(* PLC project mtcs, Institute of Astronomy Onto 0.0.1 *)
(* stored: creationDateTime 2025-03-07T11:57:23.240244, modificationDateTime 2025-03-07T11:57:23.240244 *)

TYPE MTCSParts : STRUCT
  {attribute 'TcHmiSymbol.Show'}
  telemetry : Telemetry;  (* The telemetry *)
  {attribute 'TcHmiSymbol.Show'}
  cover : Cover;  (* The Cover of the telescope *)
  {attribute 'TcHmiSymbol.Show'}
  m1 : M1;  (* The primary mirror of the telescope *)
  {attribute 'TcHmiSymbol.Show'}
  m2 : M2;  (* The secondary mirror of the telescope *)
  {attribute 'TcHmiSymbol.Show'}
  m3 : M3;  (* The tertiary mirror of the telescope *)
  {attribute 'TcHmiSymbol.Show'}
  services : Services;  (* The Services system *)
  {attribute 'TcHmiSymbol.Show'}
  safety : Safety;  (* The safety *)
  {attribute 'TcHmiSymbol.Show'}
  hydraulics : Hydraulics;  (* The hydraulics *)
  {attribute 'TcHmiSymbol.Show'}
  axes : Axes;  (* The axes *)
  {attribute 'TcHmiSymbol.Show'}
  dome : Dome;  (* The dome *)
  {attribute 'TcHmiSymbol.Show'}
  configManager : ConfigManager;  (* The config manager (to load/save/activate configuration data) *)
END_STRUCT;
END_TYPE

TYPE MTCSProcesses : STRUCT
  {attribute 'TcHmiSymbol.Show'}
  initialize : Process;  (* Start initializing the whole MTCS *)
  {attribute 'TcHmiSymbol.Show'}
  lock : Process;  (* Lock the whole MTCS *)
  {attribute 'TcHmiSymbol.Show'}
  unlock : Process;  (* Unlock the whole MTCS *)
  {attribute 'TcHmiSymbol.Show'}
  changeOperator : ChangeOperatorStateProcess;  (* Change the operator (e.g. OBSERVER, TECH, ...) *)
  {attribute 'TcHmiSymbol.Show'}
  verifyPassword : ChangeOperatorStateProcess;  (* Only verify the operator password *)
  {attribute 'TcHmiSymbol.Show'}
  reboot : Process;  (* Reboot the whole MTCS *)
  {attribute 'TcHmiSymbol.Show'}
  shutdown : Process;  (* Shutdown the whole MTCS *)
  {attribute 'TcHmiSymbol.Show'}
  wakeUp : Process;  (* Wake up the whole MTCS *)
  {attribute 'TcHmiSymbol.Show'}
  goToSleep : Process;  (* Let the whole MTCS go to sleep *)
  {attribute 'TcHmiSymbol.Show'}
  stop : Process;  (* Stop the dome and telescope *)
  {attribute 'TcHmiSymbol.Show'}
  endOfNight : Process;  (* End of night *)
  {attribute 'TcHmiSymbol.Show'}
  changeInstrument : MTCSChangeInstrumentProcess;  (* Change the instrument *)
  {attribute 'TcHmiSymbol.Show'}
  point : MTCSPointProcess;  (* Point the telescope and dome to a new target *)
  {attribute 'TcHmiSymbol.Show'}
  emergencyClose : Process;  (* Close the dome and shutter asap *)
  {attribute 'TcHmiSymbol.Show'}
  changeOperatingMode : ChangeOperatingModeStateProcess;  (* Change the operating mode (e.g. LOCAL, REMOTE, ...) *)
  {attribute 'TcHmiSymbol.Show'}
  mocsObservation : MTCSMocsObservationProcess;  (* Notifications about MOCS observation status *)
  {attribute 'TcHmiSymbol.Show'}
  remoteConnectionCheck : Process;  (* Remote connection checking *)
  {attribute 'TcHmiSymbol.Show'}
  remoteConnectionPortCheck : Process;  (* Remote connection port checking *)
  {attribute 'TcHmiSymbol.Show'}
  resetWatchdogTimer : Process;  (* Reset the watchdog timer *)
END_STRUCT;
END_TYPE

TYPE MTCSStatuses : STRUCT
  {attribute 'TcHmiSymbol.Show'}
  initializationStatus : InitializationStatus;
  {attribute 'TcHmiSymbol.Show'}
  healthStatus : HealthStatus;
  {attribute 'TcHmiSymbol.Show'}
  busyStatus : BusyStatus;
  {attribute 'TcHmiSymbol.Show'}
  operatorStatus : OperatorStatus;
  {attribute 'TcHmiSymbol.Show'}
  passwordHealthStatus : HealthStatus;
  {attribute 'TcHmiSymbol.Show'}
  activityStatus : ActivityStatus;
  {attribute 'TcHmiSymbol.Show'}
  operatingModeStatus : OperatingModeStatus;
END_STRUCT;
END_TYPE

TYPE MTCSInstrumentsConfig : STRUCT
  {attribute 'TcHmiSymbol.Show'}
  instrument0 : InstrumentConfig;  (* Instrument 0 *)
  {attribute 'TcHmiSymbol.Show'}
  instrument1 : InstrumentConfig;  (* Instrument 1 *)
  {attribute 'TcHmiSymbol.Show'}
  instrument2 : InstrumentConfig;  (* Instrument 2 *)
  {attribute 'TcHmiSymbol.Show'}
  instrument3 : InstrumentConfig;  (* Instrument 3 *)
  {attribute 'TcHmiSymbol.Show'}
  instrument4 : InstrumentConfig;  (* Instrument 4 *)
  {attribute 'TcHmiSymbol.Show'}
  instrument5 : InstrumentConfig;  (* Instrument 5 *)
  {attribute 'TcHmiSymbol.Show'}
  instrument6 : InstrumentConfig;  (* Instrument 6 *)
  {attribute 'TcHmiSymbol.Show'}
  instrument7 : InstrumentConfig;  (* Instrument 7 *)
  {attribute 'TcHmiSymbol.Show'}
  instrument8 : InstrumentConfig;  (* Instrument 8 *)
  {attribute 'TcHmiSymbol.Show'}
  instrument9 : InstrumentConfig;  (* Instrument 9 *)
END_STRUCT;
END_TYPE

TYPE MTCSEndOfNightStepConfig : STRUCT
  {attribute 'TcHmiSymbol.Show'}
  description : STRING;  (* Description of this step (to show in HMI) *)
  {attribute 'TcHmiSymbol.Show'}
  parkAxes : BOOL;  (* Park the axes *)
  {attribute 'TcHmiSymbol.Show'}
  parkAxesPosition : STRING;  (* Position to park the axes *)
  {attribute 'TcHmiSymbol.Show'}
  parkAxesWait : BOOL;  (* Wait until the axes is parked *)
  {attribute 'TcHmiSymbol.Show'}
  parkM3 : BOOL;  (* Park M3 *)
  {attribute 'TcHmiSymbol.Show'}
  parkM3Position : STRING;  (* Position to park M3 *)
  {attribute 'TcHmiSymbol.Show'}
  parkM3Wait : BOOL;  (* Wait until M3 is parked *)
  {attribute 'TcHmiSymbol.Show'}
  parkDome : BOOL;  (* Park the dome *)
  {attribute 'TcHmiSymbol.Show'}
  parkDomePosition : STRING;  (* Position to park the dome *)
  {attribute 'TcHmiSymbol.Show'}
  parkDomeWait : BOOL;  (* Wait until the dome is parked *)
  {attribute 'TcHmiSymbol.Show'}
  closeCover : BOOL;  (* Close the cover *)
  {attribute 'TcHmiSymbol.Show'}
  closeCoverWait : BOOL;  (* Wait until the cover is closed *)
  {attribute 'TcHmiSymbol.Show'}
  closeDome : BOOL;  (* Close the dome *)
  {attribute 'TcHmiSymbol.Show'}
  closeDomeWait : BOOL;  (* Wait until the dome is closed *)
  {attribute 'TcHmiSymbol.Show'}
  stop : BOOL;  (* Stop the axes and dome *)
  {attribute 'TcHmiSymbol.Show'}
  stopWait : BOOL;  (* Wait until the axes and dome are stopped *)
  {attribute 'TcHmiSymbol.Show'}
  goToSleep : BOOL;  (* Make the telescope go to sleep *)
  {attribute 'TcHmiSymbol.Show'}
  goToSleepWait : BOOL;  (* Wait until the telescope is sleeping *)
END_STRUCT;
END_TYPE

TYPE MTCSEndOfNightConfig : STRUCT
  {attribute 'TcHmiSymbol.Show'}
  step0 : MTCSEndOfNightStepConfig;  (* Step 0 *)
  {attribute 'TcHmiSymbol.Show'}
  step1 : MTCSEndOfNightStepConfig;  (* Step 1 *)
  {attribute 'TcHmiSymbol.Show'}
  step2 : MTCSEndOfNightStepConfig;  (* Step 2 *)
  {attribute 'TcHmiSymbol.Show'}
  step3 : MTCSEndOfNightStepConfig;  (* Step 3 *)
  {attribute 'TcHmiSymbol.Show'}
  step4 : MTCSEndOfNightStepConfig;  (* Step 4 *)
  {attribute 'TcHmiSymbol.Show'}
  step5 : MTCSEndOfNightStepConfig;  (* Step 5 *)
  {attribute 'TcHmiSymbol.Show'}
  step6 : MTCSEndOfNightStepConfig;  (* Step 6 *)
  {attribute 'TcHmiSymbol.Show'}
  step7 : MTCSEndOfNightStepConfig;  (* Step 7 *)
  {attribute 'TcHmiSymbol.Show'}
  step8 : MTCSEndOfNightStepConfig;  (* Step 8 *)
  {attribute 'TcHmiSymbol.Show'}
  step9 : MTCSEndOfNightStepConfig;  (* Step 9 *)
  {attribute 'TcHmiSymbol.Show'}
  step10 : MTCSEndOfNightStepConfig;  (* Step 10 *)
  {attribute 'TcHmiSymbol.Show'}
  step11 : MTCSEndOfNightStepConfig;  (* Step 11 *)
  {attribute 'TcHmiSymbol.Show'}
  step12 : MTCSEndOfNightStepConfig;  (* Step 12 *)
  {attribute 'TcHmiSymbol.Show'}
  step13 : MTCSEndOfNightStepConfig;  (* Step 13 *)
  {attribute 'TcHmiSymbol.Show'}
  step14 : MTCSEndOfNightStepConfig;  (* Step 14 *)
  {attribute 'TcHmiSymbol.Show'}
  step15 : MTCSEndOfNightStepConfig;  (* Step 15 *)
  {attribute 'TcHmiSymbol.Show'}
  step16 : MTCSEndOfNightStepConfig;  (* Step 16 *)
  {attribute 'TcHmiSymbol.Show'}
  step17 : MTCSEndOfNightStepConfig;  (* Step 17 *)
  {attribute 'TcHmiSymbol.Show'}
  step18 : MTCSEndOfNightStepConfig;  (* Step 18 *)
  {attribute 'TcHmiSymbol.Show'}
  step19 : MTCSEndOfNightStepConfig;  (* Step 19 *)
END_STRUCT;
END_TYPE

TYPE MTCSRemoteOperationConfig : STRUCT
  {attribute 'TcHmiSymbol.Show'}
  defaultOperationgMode : BOOL;  (* Default Operation Mode False=LOCAL True=REMOTE *)
  {attribute 'TcHmiSymbol.Show'}
  watchdogMocsActivityEnable : BOOL;  (* Enable the watchdog for MOCS activity *)
  {attribute 'TcHmiSymbol.Show'}
  watchdogMocsActivityTime1 : LREAL;  (* The watchdog timer time for MOCS 1 *)
  {attribute 'TcHmiSymbol.Show'}
  watchdogMocsActivityTime2 : LREAL;  (* The watchdog timer time for MOCS 2 *)
  {attribute 'TcHmiSymbol.Show'}
  warningMocsTime1 : LREAL;  (* The warning timer time for MOCS 1 *)
  {attribute 'TcHmiSymbol.Show'}
  warningMocsTime2 : LREAL;  (* The warning timer time for MOCS 2 *)
  {attribute 'TcHmiSymbol.Show'}
  watchdogRemoteConnectionEnable : BOOL;  (* Enable the watchdog for remote connection *)
  {attribute 'TcHmiSymbol.Show'}
  watchdogRemoteConnectionTime : LREAL;  (* The watchdog timer time for remote connection *)
  {attribute 'TcHmiSymbol.Show'}
  warningRemoteConnectionTime : LREAL;  (* The warning timer time for remote connection *)
  {attribute 'TcHmiSymbol.Show'}
  watchdogConnectionPortEnable : BOOL;  (* Enable the watchdog for connection Port *)
  {attribute 'TcHmiSymbol.Show'}
  watchdogConnectionPortTime : LREAL;  (* The watchdog timer time for connection Port *)
  {attribute 'TcHmiSymbol.Show'}
  warningConnectionPortTime : LREAL;  (* The warning timer time for connection Port *)
  {attribute 'TcHmiSymbol.Show'}
  remoteConnectionPortNumber : LREAL;  (* The port number for remote connection *)
END_STRUCT;
END_TYPE

TYPE MTCSConfig : STRUCT
  {attribute 'TcHmiSymbol.Show'}
  instruments : MTCSInstrumentsConfig;  (* Configure the instruments *)
  {attribute 'TcHmiSymbol.Show'}
  endOfNight : MTCSEndOfNightConfig;  (* Configure the instruments *)
  {attribute 'TcHmiSymbol.Show'}
  remoteOperation : MTCSRemoteOperationConfig;  (* Configure the remote operation *)
END_STRUCT;
END_TYPE

TYPE MTCSChangeInstrumentProcessArgs : STRUCT
  {attribute 'TcHmiSymbol.Show'}
  name : STRING;  (* Name of the instrument *)
END_STRUCT;
END_TYPE

TYPE MTCSPointProcessArgs : STRUCT
  {attribute 'TcHmiSymbol.Show'}
  alphaUnits : AxesAlphaUnits;  (* The units in which alpha is given *)
  {attribute 'TcHmiSymbol.Show'}
  alpha : LREAL;  (* Right ascention, in the units of the alphaUnits argument *)
  {attribute 'TcHmiSymbol.Show'}
  deltaUnits : AxesDeltaUnits;  (* The units in which delta is given *)
  {attribute 'TcHmiSymbol.Show'}
  delta : LREAL;  (* Declination, in the units of the deltaUnits argument *)
  {attribute 'TcHmiSymbol.Show'}
  muUnits : AxesMuUnits;  (* The units in which muAlpha and muDelta are given *)
  {attribute 'TcHmiSymbol.Show'}
  muAlpha : LREAL;  (* Right ascention proper motion, the units of muUmits (do not multiply by cos(delta)!) *)
  {attribute 'TcHmiSymbol.Show'}
  muDelta : LREAL;  (* Declination proper motion, in radians/year *)
  {attribute 'TcHmiSymbol.Show'}
  parallax : LREAL;  (* Object parallax, in arcseconds *)
  {attribute 'TcHmiSymbol.Show'}
  radialVelocity : LREAL;  (* Object radial velocity, in km/s *)
  {attribute 'TcHmiSymbol.Show'}
  epoch : LREAL := 2000.0;  (* Epoch, e.g. 2000.0 *)
  {attribute 'TcHmiSymbol.Show'}
  tracking : BOOL := TRUE;  (* True to start tracking the object, false to Only do a pointing *)
  {attribute 'TcHmiSymbol.Show'}
  rotUnits : AxesMoveUnits;  (* Units of the 'rot', 'roc' and 'ron' arguments (RADIANS, DEGREES, ARCSECONDS, ...) *)
  {attribute 'TcHmiSymbol.Show'}
  rotOffset : LREAL;  (* Offset to move the currently active rotator (incompatible with 'roc' and 'ron' args) *)
  {attribute 'TcHmiSymbol.Show'}
  rocOffset : LREAL;  (* Offset to move the cassegrain rotation axis (incompatible with 'rot' arg) *)
  {attribute 'TcHmiSymbol.Show'}
  ronOffset : LREAL;  (* Offset to move the nasmyth rotation axis (incompatible with 'rot' arg) *)
  {attribute 'TcHmiSymbol.Show'}
  doRotOffset : BOOL;  (* True to move the currently active rotator, false to leave it untouched *)
  {attribute 'TcHmiSymbol.Show'}
  doRocOffset : BOOL;  (* True to move the cassegrain rotation axis, false to leave it untouched *)
  {attribute 'TcHmiSymbol.Show'}
  doRonOffset : BOOL;  (* True to move the nasmyth rotation axis, false to leave it untouched *)
  {attribute 'TcHmiSymbol.Show'}
  doDomeTracking : BOOL := TRUE;  (* True to enable dome tracking *)
END_STRUCT;
END_TYPE

TYPE MTCSMocsObservationProcessArgs : STRUCT
  {attribute 'TcHmiSymbol.Show'}
  status : BOOL;  (* True to notify that there is an observation running *)
END_STRUCT;
END_TYPE

FUNCTION_BLOCK SM_MTCS
  VAR_INPUT
    {attribute 'TcHmiSymbol.Show'}
    {attribute 'OPC.UA.DA' := '1'}
    {attribute 'OPC.UA.DA.Access' := '1'}
    editableConfig : MTCSConfig;  (* Editable configuration of the MTCS *)
    {attribute 'TcHmiSymbol.Show'}
    {attribute 'OPC.UA.DA' := '1'}
    {attribute 'OPC.UA.DA.Access' := '1'}
    remoteOperationEnable : BOOL;  (* True to Remote operation enabled *)
    {attribute 'TcHmiSymbol.Show'}
    {attribute 'OPC.UA.DA' := '1'}
    {attribute 'OPC.UA.DA.Access' := '1'}
    mocsObservationStatus : BOOL;  (* True to notify that there is an observation running *)
    {attribute 'TcHmiSymbol.Show'}
    {attribute 'OPC.UA.DA' := '1'}
    {attribute 'OPC.UA.DA.Access' := '1'}
    remoteConnectionStatus : BOOL;  (* True to notify that there is a remote connection *)
    {attribute 'TcHmiSymbol.Show'}
    {attribute 'OPC.UA.DA' := '1'}
    {attribute 'OPC.UA.DA.Access' := '1'}
    remoteconnectionPortStatus : BOOL;  (* True to notify that there is a connection port established *)
  END_VAR
  VAR_OUTPUT
    {attribute 'OPC.UA.DA' := '1'}
    {attribute 'OPC.UA.DA.Access' := '1'}
    {attribute 'TcHmiSymbol.Show'}
    actualStatus : STRING;  (* Current status description *)
    {attribute 'TcHmiSymbol.Show'}
    previousStatus : STRING;  (* Previous status description *)
    {attribute 'TcHmiSymbol.Show'}
    {attribute 'OPC.UA.DA' := '1'}
    {attribute 'OPC.UA.DA.Access' := '1'}
    noOfFailedOperatorChanges : UINT;  (* How many times has a wrong password been entered? *)
    {attribute 'TcHmiSymbol.Show'}
    {attribute 'OPC.UA.DA' := '1'}
    {attribute 'OPC.UA.DA.Access' := '1'}
    activeInstrument : InstrumentConfig;  (* Config of the currently active instrument (depending on M3 and possibly derotator) *if* isInstrumentActive is TRUE *)
    {attribute 'TcHmiSymbol.Show'}
    {attribute 'OPC.UA.DA' := '1'}
    {attribute 'OPC.UA.DA.Access' := '1'}
    activeInstrumentNumber : INT;  (* Number of the currently active instrument (0..9, or -1 if no instrument is active) *)
    {attribute 'TcHmiSymbol.Show'}
    {attribute 'OPC.UA.DA' := '1'}
    {attribute 'OPC.UA.DA.Access' := '1'}
    activeInstrumentName : STRING;  (* Name of the currently active instrument *)
    {attribute 'TcHmiSymbol.Show'}
    {attribute 'OPC.UA.DA' := '1'}
    {attribute 'OPC.UA.DA.Access' := '1'}
    isInstrumentActive : BOOL;  (* Is an instrument currently active (i.e. is M3 static at a known position?) *)
    {attribute 'TcHmiSymbol.Show'}
    {attribute 'OPC.UA.DA' := '1'}
    {attribute 'OPC.UA.DA.Access' := '1'}
    config : MTCSConfig;  (* Active configuration of the ServicesTiming subsystem *)
    {attribute 'TcHmiSymbol.Show'}
    {attribute 'OPC.UA.DA' := '1'}
    {attribute 'OPC.UA.DA.Access' := '1'}
    remoteConnectionWarningFlag : BOOL;  (* Warning flag in case of remote connections is lost for a while *)
    {attribute 'TcHmiSymbol.Show'}
    {attribute 'OPC.UA.DA' := '1'}
    {attribute 'OPC.UA.DA.Access' := '1'}
    remoteMocsWarningFlag : BOOL;  (* Warning flag in case of there is no MOCS activity for a while *)
    {attribute 'TcHmiSymbol.Show'}
    statuses : MTCSStatuses;  (* Statuses of the state machine *)
    {attribute 'TcHmiSymbol.Show'}
    parts : MTCSParts;  (* Parts of the state machine *)
    {attribute 'TcHmiSymbol.Show'}
    processes : MTCSProcesses;  (* Processes of the state machine *)
  END_VAR

            parts.telemetry( operatorStatus := statuses.operatorStatus );
parts.cover(
    operatorStatus := statuses.operatorStatus,
    aziPos := parts.axes.parts.azi.actPos,
    elePos := parts.axes.parts.ele.actPos);
parts.m1(
    operatorStatus := statuses.operatorStatus,
    tubeAngleMeasurement := parts.telemetry.parts.accelerometers.tube);
parts.m2(
    operatorStatus := statuses.operatorStatus,
    io := parts.m1.parts.io,
    actualFocalStation := parts.m3.actualKnownPositionID,
    m3KnownPositionsConfig := parts.m3.config.knownPositions,
    temperatures := parts.telemetry.parts.temperatures);
parts.m3( operatorStatus := statuses.operatorStatus );
parts.services(
    operatorStatus := statuses.operatorStatus,
    domeApertureStatus := parts.dome.parts.shutter.statuses.apertureStatus);
parts.safety(
    operatorStatus := statuses.operatorStatus,
    activityStatus := statuses.activityStatus);
parts.hydraulics(
    operatorStatus := statuses.operatorStatus,
    safetyHydraulics := parts.safety.parts.hydraulics,
    safetyIO := parts.safety.parts.io);
parts.dome(
    operatorStatus := statuses.operatorStatus,
    activityStatus := statuses.activityStatus,
    aziTargetPos := parts.axes.parts.azi.actPos,
    safetyDomeShutter := parts.safety.parts.domeShutter,
    safetyDomeAccess := parts.safety.parts.domeAccess,
    safetyMotionBlocking := parts.safety.parts.motionBlocking);
parts.configManager( isEnabled := statuses.operatorStatus.tech );
statuses.initializationStatus();
statuses.healthStatus(
    isGood := parts.axes.statuses.healthStatus.isGood AND (parts.cover.statuses.healthStatus.isGood AND (parts.m1.statuses.healthStatus.isGood AND (parts.m2.statuses.healthStatus.isGood AND (parts.m3.statuses.healthStatus.isGood AND (parts.services.statuses.healthStatus.isGood AND (parts.telemetry.statuses.healthStatus.isGood AND (parts.safety.statuses.healthStatus.isGood AND (parts.hydraulics.statuses.healthStatus.isGood AND parts.dome.statuses.healthStatus.isGood)))))))),
    hasWarning := parts.axes.statuses.healthStatus.hasWarning OR (parts.cover.statuses.healthStatus.hasWarning OR (parts.m1.statuses.healthStatus.hasWarning OR (parts.m2.statuses.healthStatus.hasWarning OR (parts.m3.statuses.healthStatus.hasWarning OR (parts.services.statuses.healthStatus.hasWarning OR (parts.telemetry.statuses.healthStatus.hasWarning OR (parts.safety.statuses.healthStatus.hasWarning OR (parts.hydraulics.statuses.healthStatus.hasWarning OR parts.dome.statuses.healthStatus.hasWarning)))))))));
statuses.busyStatus( isBusy := parts.axes.statuses.busyStatus.busy OR (parts.cover.statuses.busyStatus.busy OR (parts.m1.statuses.busyStatus.busy OR (parts.m2.statuses.busyStatus.busy OR (parts.m3.statuses.busyStatus.busy OR (parts.services.statuses.busyStatus.busy OR (parts.telemetry.statuses.busyStatus.busy OR (parts.safety.statuses.busyStatus.busy OR (parts.hydraulics.statuses.busyStatus.busy OR parts.dome.statuses.busyStatus.busy)))))))) );
statuses.operatorStatus();
statuses.passwordHealthStatus( superState := statuses.operatorStatus.observer );
statuses.activityStatus(
    superState := statuses.initializationStatus.initialized OR statuses.initializationStatus.initializingFailed,
    isAwake := (parts.hydraulics.pumpsState = HydraulicsPumpsStates.RUNNING) OR parts.axes.statuses.poweredStatus.enabled,
    isMoving := parts.axes.statuses.busyStatus.busy OR parts.axes.isTracking);
statuses.operatingModeStatus();
processes.initialize( isEnabled := NOT(statuses.initializationStatus.initializing) );
processes.lock( isEnabled := statuses.operatorStatus.tech AND statuses.initializationStatus.initialized );
processes.unlock( isEnabled := statuses.operatorStatus.tech AND statuses.initializationStatus.locked );
processes.changeOperator( isEnabled := TRUE );
processes.verifyPassword( isEnabled := TRUE );
processes.reboot( isEnabled := TRUE );
processes.shutdown( isEnabled := statuses.operatorStatus.tech );
processes.wakeUp( isEnabled := statuses.activityStatus.sleeping );
processes.goToSleep( isEnabled := statuses.activityStatus.awake OR statuses.healthStatus.bad );
processes.stop( isEnabled := statuses.initializationStatus.initialized );
processes.endOfNight( isEnabled := TRUE );
processes.changeInstrument( isEnabled := statuses.initializationStatus.initialized OR statuses.healthStatus.bad );
processes.point( isEnabled := parts.axes.processes.point.statuses.enabledStatus.enabled AND parts.dome.processes.syncWithAxes.statuses.enabledStatus.enabled );
processes.emergencyClose( isEnabled := NOT(parts.dome.parts.shutter.statuses.apertureStatus.isClosed) );
processes.changeOperatingMode( isEnabled := statuses.operatorStatus.tech );
processes.mocsObservation( isEnabled := TRUE );
processes.remoteConnectionCheck( isEnabled := TRUE );
processes.remoteConnectionPortCheck( isEnabled := TRUE );
processes.resetWatchdogTimer( isEnabled := TRUE );

          

{attribute 'TcRpcEnable' := '1'}
METHOD initialize : RequestResults
                  initialize := THIS^.processes.initialize.request();

                
END_METHOD

{attribute 'TcRpcEnable' := '1'}
METHOD lock : RequestResults
                  lock := THIS^.processes.lock.request();

                
END_METHOD

{attribute 'TcRpcEnable' := '1'}
METHOD unlock : RequestResults
                  unlock := THIS^.processes.unlock.request();

                
END_METHOD

{attribute 'TcRpcEnable' := '1'}
METHOD changeOperator : RequestResults
  VAR_INPUT
    {attribute 'TcHmiSymbol.Show'}
    state : OperatorStates;
    {attribute 'TcHmiSymbol.Show'}
    password : STRING;
  END_VAR
                  changeOperator := THIS^.processes.changeOperator.request(
    state := state,
    password := password);

                
END_METHOD

{attribute 'TcRpcEnable' := '1'}
METHOD verifyPassword : RequestResults
  VAR_INPUT
    {attribute 'TcHmiSymbol.Show'}
    state : OperatorStates;
    {attribute 'TcHmiSymbol.Show'}
    password : STRING;
  END_VAR
                  verifyPassword := THIS^.processes.verifyPassword.request(
    state := state,
    password := password);

                
END_METHOD

{attribute 'TcRpcEnable' := '1'}
METHOD reboot : RequestResults
                  reboot := THIS^.processes.reboot.request();

                
END_METHOD

{attribute 'TcRpcEnable' := '1'}
METHOD shutdown : RequestResults
                  shutdown := THIS^.processes.shutdown.request();

                
END_METHOD

{attribute 'TcRpcEnable' := '1'}
METHOD wakeUp : RequestResults
                  wakeUp := THIS^.processes.wakeUp.request();

                
END_METHOD

{attribute 'TcRpcEnable' := '1'}
METHOD goToSleep : RequestResults
                  goToSleep := THIS^.processes.goToSleep.request();

                
END_METHOD

{attribute 'TcRpcEnable' := '1'}
METHOD stop : RequestResults
                  stop := THIS^.processes.stop.request();

                
END_METHOD

{attribute 'TcRpcEnable' := '1'}
METHOD endOfNight : RequestResults
                  endOfNight := THIS^.processes.endOfNight.request();

                
END_METHOD

{attribute 'TcRpcEnable' := '1'}
METHOD changeInstrument : RequestResults
  VAR_INPUT
    {attribute 'TcHmiSymbol.Show'}
    name : STRING;
  END_VAR
                  changeInstrument := THIS^.processes.changeInstrument.request( name := name );

                
END_METHOD

{attribute 'TcRpcEnable' := '1'}
METHOD point : RequestResults
  VAR_INPUT
    {attribute 'TcHmiSymbol.Show'}
    alphaUnits : AxesAlphaUnits;
    {attribute 'TcHmiSymbol.Show'}
    alpha : LREAL;
    {attribute 'TcHmiSymbol.Show'}
    deltaUnits : AxesDeltaUnits;
    {attribute 'TcHmiSymbol.Show'}
    delta : LREAL;
    {attribute 'TcHmiSymbol.Show'}
    muUnits : AxesMuUnits;
    {attribute 'TcHmiSymbol.Show'}
    muAlpha : LREAL;
    {attribute 'TcHmiSymbol.Show'}
    muDelta : LREAL;
    {attribute 'TcHmiSymbol.Show'}
    parallax : LREAL;
    {attribute 'TcHmiSymbol.Show'}
    radialVelocity : LREAL;
    {attribute 'TcHmiSymbol.Show'}
    epoch : LREAL;
    {attribute 'TcHmiSymbol.Show'}
    tracking : BOOL;
    {attribute 'TcHmiSymbol.Show'}
    rotUnits : AxesMoveUnits;
    {attribute 'TcHmiSymbol.Show'}
    rotOffset : LREAL;
    {attribute 'TcHmiSymbol.Show'}
    rocOffset : LREAL;
    {attribute 'TcHmiSymbol.Show'}
    ronOffset : LREAL;
    {attribute 'TcHmiSymbol.Show'}
    doRotOffset : BOOL;
    {attribute 'TcHmiSymbol.Show'}
    doRocOffset : BOOL;
    {attribute 'TcHmiSymbol.Show'}
    doRonOffset : BOOL;
    {attribute 'TcHmiSymbol.Show'}
    doDomeTracking : BOOL;
  END_VAR
                  point := THIS^.processes.point.request(
    alphaUnits := alphaUnits,
    alpha := alpha,
    deltaUnits := deltaUnits,
    delta := delta,
    muUnits := muUnits,
    muAlpha := muAlpha,
    muDelta := muDelta,
    parallax := parallax,
    radialVelocity := radialVelocity,
    epoch := epoch,
    tracking := tracking,
    rotUnits := rotUnits,
    rotOffset := rotOffset,
    rocOffset := rocOffset,
    ronOffset := ronOffset,
    doRotOffset := doRotOffset,
    doRocOffset := doRocOffset,
    doRonOffset := doRonOffset,
    doDomeTracking := doDomeTracking);

                
END_METHOD

{attribute 'TcRpcEnable' := '1'}
METHOD emergencyClose : RequestResults
                  emergencyClose := THIS^.processes.emergencyClose.request();

                
END_METHOD

{attribute 'TcRpcEnable' := '1'}
METHOD changeOperatingMode : RequestResults
  VAR_INPUT
    {attribute 'TcHmiSymbol.Show'}
    state : OperatingModeStates;
  END_VAR
                  changeOperatingMode := THIS^.processes.changeOperatingMode.request( state := state );

                
END_METHOD

{attribute 'TcRpcEnable' := '1'}
METHOD mocsObservation : RequestResults
  VAR_INPUT
    {attribute 'TcHmiSymbol.Show'}
    status : BOOL;
  END_VAR
                  mocsObservation := THIS^.processes.mocsObservation.request( status := status );

                
END_METHOD

{attribute 'TcRpcEnable' := '1'}
METHOD remoteConnectionCheck : RequestResults
                  remoteConnectionCheck := THIS^.processes.remoteConnectionCheck.request();

                
END_METHOD

{attribute 'TcRpcEnable' := '1'}
METHOD remoteConnectionPortCheck : RequestResults
                  remoteConnectionPortCheck := THIS^.processes.remoteConnectionPortCheck.request();

                
END_METHOD

{attribute 'TcRpcEnable' := '1'}
METHOD resetWatchdogTimer : RequestResults
                  resetWatchdogTimer := THIS^.processes.resetWatchdogTimer.request();

                
END_METHOD

METHOD _log : BOOL
  VAR_INPUT
    {attribute 'TcHmiSymbol.Show'}
    name : STRING;  (* Name of this function block instance *)
  END_VAR
  VAR_IN_OUT
    {attribute 'TcHmiSymbol.Show'}
    buffer : LogBuffer;  (* Buffer to write all logging to *)
  END_VAR
  VAR
    {attribute 'TcHmiSymbol.Show'}
    subBuffer : LogBuffer;  (* Temporary buffer to write logging by parts (sub-statemachines) to *)
  END_VAR
                  THIS^.parts.telemetry._log(
    name := 'telemetry',
    buffer := subBuffer);
THIS^.parts.cover._log(
    name := 'cover',
    buffer := subBuffer);
THIS^.parts.m1._log(
    name := 'm1',
    buffer := subBuffer);
THIS^.parts.m2._log(
    name := 'm2',
    buffer := subBuffer);
THIS^.parts.m3._log(
    name := 'm3',
    buffer := subBuffer);
THIS^.parts.services._log(
    name := 'services',
    buffer := subBuffer);
THIS^.parts.safety._log(
    name := 'safety',
    buffer := subBuffer);
THIS^.parts.hydraulics._log(
    name := 'hydraulics',
    buffer := subBuffer);
THIS^.parts.axes._log(
    name := 'axes',
    buffer := subBuffer);
THIS^.parts.dome._log(
    name := 'dome',
    buffer := subBuffer);
THIS^.parts.configManager._log(
    name := 'configManager',
    buffer := subBuffer);
THIS^.processes.initialize._log(
    name := 'processes.initialize',
    buffer := subBuffer);
THIS^.processes.lock._log(
    name := 'processes.lock',
    buffer := subBuffer);
THIS^.processes.unlock._log(
    name := 'processes.unlock',
    buffer := subBuffer);
THIS^.processes.changeOperator._log(
    name := 'processes.changeOperator',
    buffer := subBuffer);
THIS^.processes.verifyPassword._log(
    name := 'processes.verifyPassword',
    buffer := subBuffer);
THIS^.processes.reboot._log(
    name := 'processes.reboot',
    buffer := subBuffer);
THIS^.processes.shutdown._log(
    name := 'processes.shutdown',
    buffer := subBuffer);
THIS^.processes.wakeUp._log(
    name := 'processes.wakeUp',
    buffer := subBuffer);
THIS^.processes.goToSleep._log(
    name := 'processes.goToSleep',
    buffer := subBuffer);
THIS^.processes.stop._log(
    name := 'processes.stop',
    buffer := subBuffer);
THIS^.processes.endOfNight._log(
    name := 'processes.endOfNight',
    buffer := subBuffer);
THIS^.processes.changeInstrument._log(
    name := 'processes.changeInstrument',
    buffer := subBuffer);
THIS^.processes.point._log(
    name := 'processes.point',
    buffer := subBuffer);
THIS^.processes.emergencyClose._log(
    name := 'processes.emergencyClose',
    buffer := subBuffer);
THIS^.processes.changeOperatingMode._log(
    name := 'processes.changeOperatingMode',
    buffer := subBuffer);
THIS^.processes.mocsObservation._log(
    name := 'processes.mocsObservation',
    buffer := subBuffer);
THIS^.processes.remoteConnectionCheck._log(
    name := 'processes.remoteConnectionCheck',
    buffer := subBuffer);
THIS^.processes.remoteConnectionPortCheck._log(
    name := 'processes.remoteConnectionPortCheck',
    buffer := subBuffer);
THIS^.processes.resetWatchdogTimer._log(
    name := 'processes.resetWatchdogTimer',
    buffer := subBuffer);
LOGGER(
    name := name,
    actualStatus := THIS^.actualStatus,
    previousStatus := THIS^.previousStatus,
    buffer := buffer,
    subBuffer := subBuffer,
    pHealthStatus := ADR(THIS^.statuses.healthStatus),
    pBusyStatus := ADR(THIS^.statuses.busyStatus));

                
END_METHOD
END_FUNCTION_BLOCK

FUNCTION_BLOCK MTCSChangeInstrumentProcess EXTENDS BaseProcess
  VAR_INPUT
    {attribute 'OPC.UA.DA' := '1'}
    {attribute 'TcHmiSymbol.Show'}
    set : MTCSChangeInstrumentProcessArgs;  (* Arguments to be set, before writing do_request TRUE *)
  END_VAR
  VAR_OUTPUT
    {attribute 'OPC.UA.DA' := '1'}
    {attribute 'OPC.UA.DA.Access' := '1'}
    {attribute 'TcHmiSymbol.Show'}
    get : MTCSChangeInstrumentProcessArgs;  (* Arguments in use by the process, if do_request was accepted *)
  END_VAR

            IF do_request THEN
    do_request_result := request( name := set.name );
    do_request := FALSE;
END_IF;
SUPER^();

          

{attribute 'TcRpcEnable' := '1'}
METHOD start
  VAR_INPUT
    {attribute 'TcHmiSymbol.Show'}
    name : STRING;  (* Name of the instrument *)
  END_VAR
                  THIS^.get.name := name;
THIS^.statuses.busyStatus( isBusy := TRUE );
THIS^.statuses.healthStatus( isGood := TRUE );

                
END_METHOD

{attribute 'TcRpcEnable' := '1'}
METHOD request : RequestResults
  VAR_INPUT
    {attribute 'TcHmiSymbol.Show'}
    name : STRING;  (* Name of the instrument *)
  END_VAR
                  IF THIS^.statuses.enabledStatus.enabled THEN
    request := RequestResults.ACCEPTED;
    THIS^.start( name := name );
ELSE
    request := RequestResults.REJECTED;
END_IF;

                
END_METHOD
END_FUNCTION_BLOCK

FUNCTION_BLOCK MTCSPointProcess EXTENDS BaseProcess
  VAR_INPUT
    {attribute 'OPC.UA.DA' := '1'}
    {attribute 'TcHmiSymbol.Show'}
    set : MTCSPointProcessArgs;  (* Arguments to be set, before writing do_request TRUE *)
  END_VAR
  VAR_OUTPUT
    {attribute 'OPC.UA.DA' := '1'}
    {attribute 'OPC.UA.DA.Access' := '1'}
    {attribute 'TcHmiSymbol.Show'}
    get : MTCSPointProcessArgs;  (* Arguments in use by the process, if do_request was accepted *)
  END_VAR

            IF do_request THEN
    do_request_result := request(
    alphaUnits := set.alphaUnits,
    alpha := set.alpha,
    deltaUnits := set.deltaUnits,
    delta := set.delta,
    muUnits := set.muUnits,
    muAlpha := set.muAlpha,
    muDelta := set.muDelta,
    parallax := set.parallax,
    radialVelocity := set.radialVelocity,
    epoch := set.epoch,
    tracking := set.tracking,
    rotUnits := set.rotUnits,
    rotOffset := set.rotOffset,
    rocOffset := set.rocOffset,
    ronOffset := set.ronOffset,
    doRotOffset := set.doRotOffset,
    doRocOffset := set.doRocOffset,
    doRonOffset := set.doRonOffset,
    doDomeTracking := set.doDomeTracking);
    do_request := FALSE;
END_IF;
SUPER^();

          

{attribute 'TcRpcEnable' := '1'}
METHOD start
  VAR_INPUT
    {attribute 'TcHmiSymbol.Show'}
    alphaUnits : AxesAlphaUnits;  (* The units in which alpha is given *)
    {attribute 'TcHmiSymbol.Show'}
    alpha : LREAL;  (* Right ascention, in the units of the alphaUnits argument *)
    {attribute 'TcHmiSymbol.Show'}
    deltaUnits : AxesDeltaUnits;  (* The units in which delta is given *)
    {attribute 'TcHmiSymbol.Show'}
    delta : LREAL;  (* Declination, in the units of the deltaUnits argument *)
    {attribute 'TcHmiSymbol.Show'}
    muUnits : AxesMuUnits;  (* The units in which muAlpha and muDelta are given *)
    {attribute 'TcHmiSymbol.Show'}
    muAlpha : LREAL;  (* Right ascention proper motion, the units of muUmits (do not multiply by cos(delta)!) *)
    {attribute 'TcHmiSymbol.Show'}
    muDelta : LREAL;  (* Declination proper motion, in radians/year *)
    {attribute 'TcHmiSymbol.Show'}
    parallax : LREAL;  (* Object parallax, in arcseconds *)
    {attribute 'TcHmiSymbol.Show'}
    radialVelocity : LREAL;  (* Object radial velocity, in km/s *)
    {attribute 'TcHmiSymbol.Show'}
    epoch : LREAL := 2000.0;  (* Epoch, e.g. 2000.0 *)
    {attribute 'TcHmiSymbol.Show'}
    tracking : BOOL := TRUE;  (* True to start tracking the object, false to Only do a pointing *)
    {attribute 'TcHmiSymbol.Show'}
    rotUnits : AxesMoveUnits;  (* Units of the 'rot', 'roc' and 'ron' arguments (RADIANS, DEGREES, ARCSECONDS, ...) *)
    {attribute 'TcHmiSymbol.Show'}
    rotOffset : LREAL;  (* Offset to move the currently active rotator (incompatible with 'roc' and 'ron' args) *)
    {attribute 'TcHmiSymbol.Show'}
    rocOffset : LREAL;  (* Offset to move the cassegrain rotation axis (incompatible with 'rot' arg) *)
    {attribute 'TcHmiSymbol.Show'}
    ronOffset : LREAL;  (* Offset to move the nasmyth rotation axis (incompatible with 'rot' arg) *)
    {attribute 'TcHmiSymbol.Show'}
    doRotOffset : BOOL;  (* True to move the currently active rotator, false to leave it untouched *)
    {attribute 'TcHmiSymbol.Show'}
    doRocOffset : BOOL;  (* True to move the cassegrain rotation axis, false to leave it untouched *)
    {attribute 'TcHmiSymbol.Show'}
    doRonOffset : BOOL;  (* True to move the nasmyth rotation axis, false to leave it untouched *)
    {attribute 'TcHmiSymbol.Show'}
    doDomeTracking : BOOL := TRUE;  (* True to enable dome tracking *)
  END_VAR
                  THIS^.get.alphaUnits := alphaUnits;
THIS^.get.alpha := alpha;
THIS^.get.deltaUnits := deltaUnits;
THIS^.get.delta := delta;
THIS^.get.muUnits := muUnits;
THIS^.get.muAlpha := muAlpha;
THIS^.get.muDelta := muDelta;
THIS^.get.parallax := parallax;
THIS^.get.radialVelocity := radialVelocity;
THIS^.get.epoch := epoch;
THIS^.get.tracking := tracking;
THIS^.get.rotUnits := rotUnits;
THIS^.get.rotOffset := rotOffset;
THIS^.get.rocOffset := rocOffset;
THIS^.get.ronOffset := ronOffset;
THIS^.get.doRotOffset := doRotOffset;
THIS^.get.doRocOffset := doRocOffset;
THIS^.get.doRonOffset := doRonOffset;
THIS^.get.doDomeTracking := doDomeTracking;
THIS^.statuses.busyStatus( isBusy := TRUE );
THIS^.statuses.healthStatus( isGood := TRUE );

                
END_METHOD

{attribute 'TcRpcEnable' := '1'}
METHOD request : RequestResults
  VAR_INPUT
    {attribute 'TcHmiSymbol.Show'}
    alphaUnits : AxesAlphaUnits;  (* The units in which alpha is given *)
    {attribute 'TcHmiSymbol.Show'}
    alpha : LREAL;  (* Right ascention, in the units of the alphaUnits argument *)
    {attribute 'TcHmiSymbol.Show'}
    deltaUnits : AxesDeltaUnits;  (* The units in which delta is given *)
    {attribute 'TcHmiSymbol.Show'}
    delta : LREAL;  (* Declination, in the units of the deltaUnits argument *)
    {attribute 'TcHmiSymbol.Show'}
    muUnits : AxesMuUnits;  (* The units in which muAlpha and muDelta are given *)
    {attribute 'TcHmiSymbol.Show'}
    muAlpha : LREAL;  (* Right ascention proper motion, the units of muUmits (do not multiply by cos(delta)!) *)
    {attribute 'TcHmiSymbol.Show'}
    muDelta : LREAL;  (* Declination proper motion, in radians/year *)
    {attribute 'TcHmiSymbol.Show'}
    parallax : LREAL;  (* Object parallax, in arcseconds *)
    {attribute 'TcHmiSymbol.Show'}
    radialVelocity : LREAL;  (* Object radial velocity, in km/s *)
    {attribute 'TcHmiSymbol.Show'}
    epoch : LREAL := 2000.0;  (* Epoch, e.g. 2000.0 *)
    {attribute 'TcHmiSymbol.Show'}
    tracking : BOOL := TRUE;  (* True to start tracking the object, false to Only do a pointing *)
    {attribute 'TcHmiSymbol.Show'}
    rotUnits : AxesMoveUnits;  (* Units of the 'rot', 'roc' and 'ron' arguments (RADIANS, DEGREES, ARCSECONDS, ...) *)
    {attribute 'TcHmiSymbol.Show'}
    rotOffset : LREAL;  (* Offset to move the currently active rotator (incompatible with 'roc' and 'ron' args) *)
    {attribute 'TcHmiSymbol.Show'}
    rocOffset : LREAL;  (* Offset to move the cassegrain rotation axis (incompatible with 'rot' arg) *)
    {attribute 'TcHmiSymbol.Show'}
    ronOffset : LREAL;  (* Offset to move the nasmyth rotation axis (incompatible with 'rot' arg) *)
    {attribute 'TcHmiSymbol.Show'}
    doRotOffset : BOOL;  (* True to move the currently active rotator, false to leave it untouched *)
    {attribute 'TcHmiSymbol.Show'}
    doRocOffset : BOOL;  (* True to move the cassegrain rotation axis, false to leave it untouched *)
    {attribute 'TcHmiSymbol.Show'}
    doRonOffset : BOOL;  (* True to move the nasmyth rotation axis, false to leave it untouched *)
    {attribute 'TcHmiSymbol.Show'}
    doDomeTracking : BOOL := TRUE;  (* True to enable dome tracking *)
  END_VAR
                  IF THIS^.statuses.enabledStatus.enabled THEN
    request := RequestResults.ACCEPTED;
    THIS^.start(
        alphaUnits := alphaUnits,
        alpha := alpha,
        deltaUnits := deltaUnits,
        delta := delta,
        muUnits := muUnits,
        muAlpha := muAlpha,
        muDelta := muDelta,
        parallax := parallax,
        radialVelocity := radialVelocity,
        epoch := epoch,
        tracking := tracking,
        rotUnits := rotUnits,
        rotOffset := rotOffset,
        rocOffset := rocOffset,
        ronOffset := ronOffset,
        doRotOffset := doRotOffset,
        doRocOffset := doRocOffset,
        doRonOffset := doRonOffset,
        doDomeTracking := doDomeTracking);
ELSE
    request := RequestResults.REJECTED;
END_IF;

                
END_METHOD
END_FUNCTION_BLOCK

FUNCTION_BLOCK MTCSMocsObservationProcess EXTENDS BaseProcess
  VAR_INPUT
    {attribute 'OPC.UA.DA' := '1'}
    {attribute 'TcHmiSymbol.Show'}
    set : MTCSMocsObservationProcessArgs;  (* Arguments to be set, before writing do_request TRUE *)
  END_VAR
  VAR_OUTPUT
    {attribute 'OPC.UA.DA' := '1'}
    {attribute 'OPC.UA.DA.Access' := '1'}
    {attribute 'TcHmiSymbol.Show'}
    get : MTCSMocsObservationProcessArgs;  (* Arguments in use by the process, if do_request was accepted *)
  END_VAR

            IF do_request THEN
    do_request_result := request( status := set.status );
    do_request := FALSE;
END_IF;
SUPER^();

          

{attribute 'TcRpcEnable' := '1'}
METHOD start
  VAR_INPUT
    {attribute 'TcHmiSymbol.Show'}
    status : BOOL;  (* True to notify that there is an observation running *)
  END_VAR
                  THIS^.get.status := status;
THIS^.statuses.busyStatus( isBusy := TRUE );
THIS^.statuses.healthStatus( isGood := TRUE );

                
END_METHOD

{attribute 'TcRpcEnable' := '1'}
METHOD request : RequestResults
  VAR_INPUT
    {attribute 'TcHmiSymbol.Show'}
    status : BOOL;  (* True to notify that there is an observation running *)
  END_VAR
                  IF THIS^.statuses.enabledStatus.enabled THEN
    request := RequestResults.ACCEPTED;
    THIS^.start( status := status );
ELSE
    request := RequestResults.REJECTED;
END_IF;

                
END_METHOD
END_FUNCTION_BLOCK
